FUNCTION_BLOCK FB_LiftB EXTENDS FB_Lift
VAR_INPUT
END_VAR
VAR_OUTPUT
END_VAR
VAR
END_VAR

END_FUNCTION_BLOCK

(* stored: Version 1.1.0.1
   POU FB_LiftB: Id {2a47a6c6-b1e5-452f-b183-c91f9828a8a6}, SpecialFunc None *)
